Fanuc KAREL source: NC0001.KL

-- PROVISIONAL review KL for V1013-1; original PC SHA256 44238abc31c5ab4ed42b5fcef69f822fd8c7022ab6c27570b6dd30f1e248b2c2
-- Incomplete behavior may be omitted. Consult companion uncertainty JSON. Do not deploy.
PROGRAM NC0001
%NOLOCKGROUP
-- UNRESOLVED_LOCAL_POOL 1 cells at code offset 3; source declarations unknown
-- DIRECT_LOCAL_WORD_ACCESS alone does not prove INTEGER, REAL, or BOOLEAN
BEGIN
  -- UNRESOLVED_PC offsets 0-8; opcodes 2B,2C,7B
  -- UNRESOLVED_PC offsets 13-20; opcodes 9D,23
  -- UNRESOLVED_PC offsets 25-39; opcodes 21,9D,52,23
  -- UNRESOLVED_PC offsets 44-48; opcodes 7F
  -- UNRESOLVED_PC offsets 53-57; opcodes 27,AA
  -- UNRESOLVED_PC offsets 62-66; opcodes 7F
END NC0001
